KUKA KRL program: ps_p13060r5_msr_lta_c1.src, ps_p13060r5_msr_lta_c1.dat

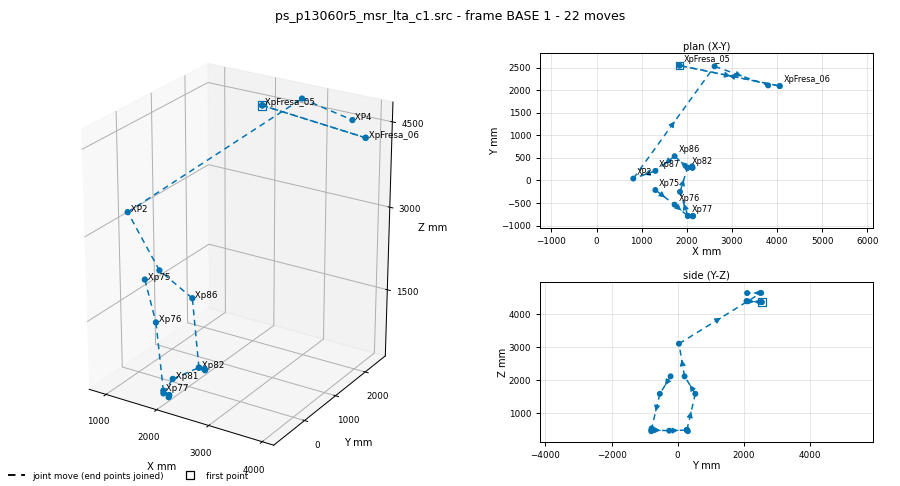
[picture p0: tool path of ps_p13060r5_msr_lta_c1.src in frame BASE 1, 22 of 24 moves have a stored position in this frame; points joined in program order, loops and branches not executed]
--- ps_p13060r5_msr_lta_c1.src ---
&ACCESS RVO
&REL 5
&COMMENT SOLDA MSR LTA GUN C1
&PARAM DISKPATH = KRC:\R1\Program
DEF ps_p13060r5_msr_lta_c1( )
;FOLD INI
  ;FOLD BASISTECH INI
    GLOBAL INTERRUPT DECL 3 WHEN $STOPMESS==TRUE DO IR_STOPM ( )
    INTERRUPT ON 3
    BAS (#INITMOV,0 )
  ;ENDFOLD (BASISTECH INI)
;FOLD SPOTTECH INI
USERSPOT(#INIT)
;ENDFOLD (SPOTTECH INI)
;FOLD GRIPPERTECH INI

;ENDFOLD (GRIPPERTECH INI)
  ;FOLD USER INI
    ;Make your modifications here

     ;FOLD COLLISION_V_3.01 INI ;%{E}
        IF (COLLISION_DATA[1].I_NR>0) THEN
          GLOBAL INTERRUPT DECL 21 WHEN $IN[COLLISION_DATA[1].I_NR]==FALSE DO COLLSTOP (1,0 )
        ENDIF
        IF (COLLISION_DATA[2].I_NR>0) THEN
          GLOBAL INTERRUPT DECL 22 WHEN $IN[COLLISION_DATA[2].I_NR]==FALSE DO COLLSTOP (2,0 )
        ENDIF
        IF (COLLISION_DATA[3].I_NR>0) THEN
          GLOBAL INTERRUPT DECL 23 WHEN $IN[COLLISION_DATA[3].I_NR]==FALSE DO COLLSTOP (3,0 )
        ENDIF
        IF (COLLISION_DATA[4].I_NR>0) THEN
          GLOBAL INTERRUPT DECL 24 WHEN $IN[COLLISION_DATA[4].I_NR]==FALSE DO COLLSTOP (4,0 )
        ENDIF
     ;ENDFOLD (Collision)

  ;ENDFOLD (USER INI)
;ENDFOLD (INI)

; Caracterização dos meios de produção: P13.060-R5
; Versão atual: 17/07/2013 Nome: Solda C1
; Change: MGS/LTA

chk_w2_wechs_ok ( )           ; VERIFICAÇÃO DE FERRAMENA: C1

;FOLD PTP HOME2 Vel=100 % DEFAULT;%{PE}%R 8.2.20,%MKUKATPBASIS,%CMOVE,%VPTP,%P 1:PTP, 2:HOME2, 3:, 5:100, 7:DEFAULT
$BWDSTART=FALSE
PDAT_ACT=PDEFAULT
FDAT_ACT=FHOME2
BAS(#PTP_PARAMS,100)
PTP XHOME2
;ENDFOLD

IF MaxStandMenge (1) THEN
 MaxStandmengeErreicht (1)
ENDIF

IF Elektrodenwechsel (1) THEN
;FOLD PTP pFresa_05 CONT Vel=100 % PDAT4 Tool[2]:Gun C1 Base[1]:Actros;%{PE}%R 8.2.20,%MKUKATPBASIS,%CMOVE,%VPTP,%P 1:PTP, 2:pFresa_05, 3:C_DIS, 5:100, 7:PDAT4
$BWDSTART=FALSE
PDAT_ACT=PPDAT4
FDAT_ACT=FpFresa_05
BAS(#PTP_PARAMS,100)
PTP XpFresa_05 C_DIS
;ENDFOLD
;FOLD PULSE 168 'DOCK 1 Fechar Proteção' State=TRUE Time=1 sec;%{PE}%R 8.2.20,%MKUKATPBASIS,%COUT,%VPULSE,%P 2:168, 3:DOCK 1 Fechar Proteção, 5:TRUE, 6:, 8:1
PULSE($OUT[168], TRUE,1)
;ENDFOLD
;FOLD WAIT FOR ( IN 166 'DOCK 1 Proteção Fechada' );%{PE}%R 8.2.20,%MKUKATPBASIS,%CEXT_WAIT_FOR,%VEXT_WAIT_FOR,%P 2:, 4:, 5:$IN, 6:166, 7:DOCK 1 Proteção Fechada, 9:
WAIT FOR  ( $IN[166] )
;ENDFOLD
;FOLD PTP pFresa_06 CONT Vel=100 % PDAT5 Tool[2]:Gun C1 Base[1]:Actros;%{PE}%R 8.2.20,%MKUKATPBASIS,%CMOVE,%VPTP,%P 1:PTP, 2:pFresa_06, 3:C_DIS, 5:100, 7:PDAT5
$BWDSTART=FALSE
PDAT_ACT=PPDAT5
FDAT_ACT=FpFresa_06
BAS(#PTP_PARAMS,100)
PTP XpFresa_06 C_DIS
;ENDFOLD
 e_Fraes_2 ()
;FOLD PTP pFresa_07 CONT Vel=100 % PDAT6 Tool[2]:Gun C1 Base[1]:Actros;%{PE}%R 8.2.20,%MKUKATPBASIS,%CMOVE,%VPTP,%P 1:PTP, 2:pFresa_07, 3:C_DIS, 5:100, 7:PDAT6
$BWDSTART=FALSE
PDAT_ACT=PPDAT6
FDAT_ACT=FpFresa_07
BAS(#PTP_PARAMS,100)
PTP XpFresa_07 C_DIS
;ENDFOLD
;FOLD PTP pFresa_08 CONT Vel=100 % PDAT7 Tool[2]:Gun C1 Base[1]:Actros;%{PE}%R 8.2.20,%MKUKATPBASIS,%CMOVE,%VPTP,%P 1:PTP, 2:pFresa_08, 3:C_DIS, 5:100, 7:PDAT7
$BWDSTART=FALSE
PDAT_ACT=PPDAT7
FDAT_ACT=FpFresa_08
BAS(#PTP_PARAMS,100)
PTP XpFresa_08 C_DIS
;ENDFOLD
ENDIF

;FOLD PTP HOME2 Vel=100 % DEFAULT;%{PE}%R 8.2.20,%MKUKATPBASIS,%CMOVE,%VPTP,%P 1:PTP, 2:HOME2, 3:, 5:100, 7:DEFAULT
$BWDSTART=FALSE
PDAT_ACT=PDEFAULT
FDAT_ACT=FHOME2
BAS(#PTP_PARAMS,100)
PTP XHOME2
;ENDFOLD

;FOLD OUT 3339 'R5 SOLDANDO' State=FALSE ;%{PE}%R 8.2.20,%MKUKATPBASIS,%COUT,%VOUTX,%P 2:3339, 3:R5 SOLDANDO, 5:FALSE, 6:
$OUT[3339]=FALSE
;ENDFOLD

;FOLD PTP p75 CONT Vel=100 % P_OLP2 Tool[2]:Gun C1 Base[1]:Actros;%{PE}%R 8.2.20,%MKUKATPBASIS,%CMOVE,%VPTP,%P 1:PTP, 2:p75, 3:C_DIS, 5:100, 7:P_OLP2
$BWDSTART=FALSE
PDAT_ACT=PP_OLP2
FDAT_ACT=Fp75
BAS(#PTP_PARAMS,100)
PTP Xp75 C_DIS
;ENDFOLD
;FOLD PTP p76 CONT Vel=100 % P_OLP3 Tool[2]:Gun C1 Base[1]:Actros;%{PE}%R8.2,%MKUKATPBASIS,%CMOVE,%VPTP,%P 1:PTP, 2:p76, 3:C_DIS, 5:100, 7:P_OLP3
$BWDSTART = FALSE
PDAT_ACT= PP_OLP3
FDAT_ACT= Fp76
BAS(#PTP_PARAMS,100)
PTP Xp76 C_DIS
;ENDFOLD
;FOLD PTP p77 CONT Vel=100 % P_OLP4 Tool[2]:Gun C1 Base[1]:Actros;%{PE}%R8.2,%MKUKATPBASIS,%CMOVE,%VPTP,%P 1:PTP, 2:p77, 3:C_DIS, 5:100, 7:P_OLP4
$BWDSTART = FALSE
PDAT_ACT= PP_OLP4
FDAT_ACT= Fp77
BAS(#PTP_PARAMS,100)
PTP Xp77 C_DIS
;ENDFOLD
;FOLD PTP p78 CONT Vel=100 % P_OLP5 Tool[2]:Gun C1 Base[1]:Actros;%{PE}%R8.2,%MKUKATPBASIS,%CMOVE,%VPTP,%P 1:PTP, 2:p78, 3:C_DIS, 5:100, 7:P_OLP5
$BWDSTART = FALSE
PDAT_ACT= PP_OLP5
FDAT_ACT= Fp78
BAS(#PTP_PARAMS,100)
PTP Xp78 C_DIS
;ENDFOLD

;FOLD ; SWP_60_5471;%{PE}%R8.2,%MKUKATPBASIS,%CCOMMENT,%VNORMAL,%P 2: SWP_60_5471
;ENDFOLD
;FOLD PTP swp_60_5471 P_OLP6 SPOT Gun=1 RETR OPN PgNo1=55 ACTIVE=1 Tool[2]:Gun C1 Base[1]:Actros;%{PE}%R 8.2.2,%MKUKATPSPOT,%CSPOT,%VPTP,%P 1:PTP, 2:swp_60_5471, 3:, 5:100, 7:P_OLP6, 10:1, 12:#FIRST, 14:#OPN, 16:55, 18:1, 20:1, 22:0, 24:1, 25:S_OLP1
$BWDSTART=FALSE
PDAT_ACT=PP_OLP6
FDAT_ACT=Fswp_60_5471
BAS(#PTP_PARAMS,PP_OLP6.VEL)
S_ACT.GUN=1
S_ACT.PAIR=SDEFAULT.PAIR
S_ACT.RETR=#OPN
S_ACT.CLO_TM=1
S_ACT.PGNO1=55
S_ACT.PGNO2=SDEFAULT.PGNO2
S_ACT.PRESS1=SDEFAULT.PRESS1
S_ACT.PRESS2=SDEFAULT.PRESS2
S_READY=FALSE
PTP Xswp_60_5471
USERSPOT(#SPOT, S_ACT)
WAIT FOR S_READY
;ENDFOLD

;FOLD PTP p79 CONT Vel=100 % P_OLP7 Tool[2]:Gun C1 Base[1]:Actros;%{PE}%R8.2,%MKUKATPBASIS,%CMOVE,%VPTP,%P 1:PTP, 2:p79, 3:C_DIS, 5:100, 7:P_OLP7
$BWDSTART = FALSE
PDAT_ACT= PP_OLP7
FDAT_ACT= Fp79
BAS(#PTP_PARAMS,100)
PTP Xp79 C_DIS
;ENDFOLD
;FOLD PTP p80 CONT Vel=100 % P_OLP8 Tool[2]:Gun C1 Base[1]:Actros;%{PE}%R8.2,%MKUKATPBASIS,%CMOVE,%VPTP,%P 1:PTP, 2:p80, 3:C_DIS, 5:100, 7:P_OLP8
$BWDSTART = FALSE
PDAT_ACT= PP_OLP8
FDAT_ACT= Fp80
BAS(#PTP_PARAMS,100)
PTP Xp80 C_DIS
;ENDFOLD
;FOLD PTP p81 CONT Vel=100 % P_OLP9 Tool[2]:Gun C1 Base[1]:Actros;%{PE}%R8.2,%MKUKATPBASIS,%CMOVE,%VPTP,%P 1:PTP, 2:p81, 3:C_DIS, 5:100, 7:P_OLP9
$BWDSTART = FALSE
PDAT_ACT= PP_OLP9
FDAT_ACT= Fp81
BAS(#PTP_PARAMS,100)
PTP Xp81 C_DIS
;ENDFOLD
;FOLD PTP p82 CONT Vel=100 % P_OLP10 Tool[2]:Gun C1 Base[1]:Actros;%{PE}%R8.2,%MKUKATPBASIS,%CMOVE,%VPTP,%P 1:PTP, 2:p82, 3:C_DIS, 5:100, 7:P_OLP10
$BWDSTART = FALSE
PDAT_ACT= PP_OLP10
FDAT_ACT= Fp82
BAS(#PTP_PARAMS,100)
PTP Xp82 C_DIS
;ENDFOLD
;FOLD PTP p83 CONT Vel=100 % P_OLP11 Tool[2]:Gun C1 Base[1]:Actros;%{PE}%R8.2,%MKUKATPBASIS,%CMOVE,%VPTP,%P 1:PTP, 2:p83, 3:C_DIS, 5:100, 7:P_OLP11
$BWDSTART = FALSE
PDAT_ACT= PP_OLP11
FDAT_ACT= Fp83
BAS(#PTP_PARAMS,100)
PTP Xp83 C_DIS
;ENDFOLD

;FOLD ; SWP_60_5452;%{PE}%R8.2,%MKUKATPBASIS,%CCOMMENT,%VNORMAL,%P 2: SWP_60_5452
;ENDFOLD
;FOLD PTP swp_60_5452 P_OLP12 SPOT Gun=1 RETR OPN PgNo1=56 ACTIVE=1 Tool[2]:Gun C1 Base[1]:Actros;%{PE}%R 8.2.2,%MKUKATPSPOT,%CSPOT,%VPTP,%P 1:PTP, 2:swp_60_5452, 3:, 5:100, 7:P_OLP12, 10:1, 12:#FIRST, 14:#OPN, 16:56, 18:1, 20:1, 22:0, 24:1, 25:S_OLP2
$BWDSTART=FALSE
PDAT_ACT=PP_OLP12
FDAT_ACT=Fswp_60_5452
BAS(#PTP_PARAMS,PP_OLP12.VEL)
S_ACT.GUN=1
S_ACT.PAIR=SDEFAULT.PAIR
S_ACT.RETR=#OPN
S_ACT.CLO_TM=1
S_ACT.PGNO1=56
S_ACT.PGNO2=SDEFAULT.PGNO2
S_ACT.PRESS1=SDEFAULT.PRESS1
S_ACT.PRESS2=SDEFAULT.PRESS2
S_READY=FALSE
PTP Xswp_60_5452
USERSPOT(#SPOT, S_ACT)
WAIT FOR S_READY
;ENDFOLD

;FOLD PTP p84 CONT Vel=100 % P_OLP13 Tool[2]:Gun C1 Base[1]:Actros;%{PE}%R8.2,%MKUKATPBASIS,%CMOVE,%VPTP,%P 1:PTP, 2:p84, 3:C_DIS, 5:100, 7:P_OLP13
$BWDSTART = FALSE
PDAT_ACT= PP_OLP13
FDAT_ACT= Fp84
BAS(#PTP_PARAMS,100)
PTP Xp84 C_DIS
;ENDFOLD
;FOLD PTP p85 CONT Vel=100 % P_OLP14 Tool[2]:Gun C1 Base[1]:Actros;%{PE}%R8.2,%MKUKATPBASIS,%CMOVE,%VPTP,%P 1:PTP, 2:p85, 3:C_DIS, 5:100, 7:P_OLP14
$BWDSTART = FALSE
PDAT_ACT= PP_OLP14
FDAT_ACT= Fp85
BAS(#PTP_PARAMS,100)
PTP Xp85 C_DIS
;ENDFOLD
;FOLD PTP p86 CONT Vel=100 % P_OLP15 Tool[2]:Gun C1 Base[1]:Actros;%{PE}%R8.2,%MKUKATPBASIS,%CMOVE,%VPTP,%P 1:PTP, 2:p86, 3:C_DIS, 5:100, 7:P_OLP15
$BWDSTART = FALSE
PDAT_ACT= PP_OLP15
FDAT_ACT= Fp86
BAS(#PTP_PARAMS,100)
PTP Xp86 C_DIS
;ENDFOLD
;FOLD PTP p87 CONT Vel=100 % P_OLP16 Tool[2]:Gun C1 Base[1]:Actros;%{PE}%R8.2,%MKUKATPBASIS,%CMOVE,%VPTP,%P 1:PTP, 2:p87, 3:C_DIS, 5:100, 7:P_OLP16
$BWDSTART = FALSE
PDAT_ACT= PP_OLP16
FDAT_ACT= Fp87
BAS(#PTP_PARAMS,100)
PTP Xp87 C_DIS
;ENDFOLD

;FOLD OUT 3339 'R5 SOLDANDO' State=TRUE CONT;%{PE}%R 8.2.20,%MKUKATPBASIS,%COUT,%VOUTX,%P 2:3339, 3:R5 SOLDANDO, 5:TRUE, 6:CONTINUE
CONTINUE
$OUT[3339]=TRUE
;ENDFOLD

;FOLD PTP P2 CONT Vel=100 % PDAT2 Tool[2]:Gun C1 Base[1]:Actros;%{PE}%R 8.2.20,%MKUKATPBASIS,%CMOVE,%VPTP,%P 1:PTP, 2:P2, 3:C_DIS, 5:100, 7:PDAT2
$BWDSTART=FALSE
PDAT_ACT=PPDAT2
FDAT_ACT=FP2
BAS(#PTP_PARAMS,100)
PTP XP2 C_DIS
;ENDFOLD
;FOLD PTP P3 CONT Vel=100 % PDAT3 Tool[2]:Gun C1 Base[1]:Actros;%{PE}%R 8.2.20,%MKUKATPBASIS,%CMOVE,%VPTP,%P 1:PTP, 2:P3, 3:C_DIS, 5:100, 7:PDAT3
$BWDSTART=FALSE
PDAT_ACT=PPDAT3
FDAT_ACT=FP3
BAS(#PTP_PARAMS,100)
PTP XP3 C_DIS
;ENDFOLD
;FOLD PTP P4 Vel=100 % PDAT8 Tool[2]:Gun C1 Base[1]:Actros;%{PE}%R 8.2.20,%MKUKATPBASIS,%CMOVE,%VPTP,%P 1:PTP, 2:P4, 3:, 5:100, 7:PDAT8
$BWDSTART=FALSE
PDAT_ACT=PPDAT8
FDAT_ACT=FP4
BAS(#PTP_PARAMS,100)
PTP XP4
;ENDFOLD

IF FraesAnf (1) THEN

 f_Fraes_2()

ENDIF

END

--- ps_p13060r5_msr_lta_c1.dat ---
&ACCESS RVO
&REL 5
&COMMENT SOLDA MSR LTA GUN C1
&PARAM DISKPATH = KRC:\R1\Program
DEFDAT  ps_p13060r5_msr_lta_c1
;FOLD EXTERNAL DECLARATIONS;%{PE}%MKUKATPBASIS,%CEXT,%VCOMMON,%P
;FOLD GRIPPERTECH EXT
EXT  H50 (INT  :IN,INT  :IN,INT  :IN,GRP_TYP  :IN )
;ENDFOLD (GRIPPERTECH EXT)
;FOLD SPOTTECH EXT
EXT  USERSPOT (S_COMMAND  :IN,SPOT_TYPE  :IN )
;ENDFOLD (SPOTTECH EXT)
;FOLD BASISTECH EXT;%{PE}%MKUKATPBASIS,%CEXT,%VEXT,%P
EXT  BAS (BAS_COMMAND  :IN,REAL  :IN )
DECL INT SUCCESS
;ENDFOLD (BASISTECH EXT)
;FOLD USER EXT;%{E}%MKUKATPUSER,%CEXT,%VEXT,%P
;Make your modifications here

;ENDFOLD (USER EXT)
;ENDFOLD (EXTERNAL DECLARATIONS)

;# ============ START PATH : swp_p13060r5_msr_lta_c1 =============
DECL FDAT Fp75={TOOL_NO 2,BASE_NO 1,IPO_FRAME #BASE,POINT2[] " "}
DECL PDAT PP_OLP2={VEL 100.0,ACC 100.0,APO_DIST 100.0,APO_MODE #CDIS}
DECL E6POS Xp75={X 1303.604,Y -211.761002,Z 2118.72705,A -126.906303,B 65.6848984,C 49.8302002,S 2,T 10}
DECL FDAT Fp76={TOOL_NO 2,BASE_NO 1,IPO_FRAME #BASE,POINT2[] " "}
DECL PDAT PP_OLP3={VEL 100.0,ACC 100.0,APO_DIST 100.0,APO_MODE #CDIS}
DECL E6POS Xp76={X 1729.96497,Y -537.172974,Z 1590.30103,A -75.8211975,B 62.4005013,C 105.7089,S 2,T 11}
DECL FDAT Fp77={TOOL_NO 2,BASE_NO 1,IPO_FRAME #BASE,POINT2[] " "}
DECL PDAT PP_OLP4={VEL 100.0,ACC 100.0,APO_DIST 100.0,APO_MODE #CDIS}
DECL E6POS Xp77={X 2022.47803,Y -785.769104,Z 542.154907,A -89.9998932,B 70.0002136,C 89.9999771,S 2,T 9,E1 0.0,E2 0.0,E3 0.0,E4 0.0,E5 0.0,E6 0.0}
DECL FDAT Fp78={TOOL_NO 2,BASE_NO 1,IPO_FRAME #BASE,POINT2[] " "}
DECL PDAT PP_OLP5={VEL 100.0,ACC 100.0,APO_DIST 100.0,APO_MODE #CDIS}
DECL E6POS Xp78={X 2134.76611,Y -787.281006,Z 490.900208,A -89.9603119,B 69.9023438,C 90.0867233,S 2,T 9,E1 0.0,E2 0.0,E3 0.0,E4 0.0,E5 0.0,E6 0.0}
DECL FDAT Fswp_60_5471={TOOL_NO 2,BASE_NO 1,IPO_FRAME #BASE,POINT2[] " "}
DECL PDAT PP_OLP6={VEL 100.0,ACC 100.0,APO_DIST 0.0}
DECL SPOT_TYPE SS_OLP1={GUN 2,PAIR #FIRST,RETR #CLO,CLO_TM 0,PGNO1 1,PRESS1 1.0,PGNO2 0,PRESS2 0.0}
DECL E6POS Xswp_60_5471={X 2130.88208,Y -795.672913,Z 457.943512,A -90.164978,B 69.9813766,C 89.8283234,S 2,T 9,E1 0.0,E2 0.0,E3 0.0,E4 0.0,E5 0.0,E6 0.0}
DECL FDAT Fp79={TOOL_NO 2,BASE_NO 1,IPO_FRAME #BASE,POINT2[] " "}
DECL PDAT PP_OLP7={VEL 100.0,ACC 100.0,APO_DIST 100.0,APO_MODE #CDIS}
DECL E6POS Xp79={X 2134.00098,Y -785.97699,Z 492.528015,A -90.0,B 70.0,C 90.0,S 2,T 9,E1 0.0,E2 0.0,E3 0.0,E4 0.0,E5 0.0,E6 0.0}
DECL FDAT Fp80={TOOL_NO 2,BASE_NO 1,IPO_FRAME #BASE,POINT2[] " "}
DECL PDAT PP_OLP8={VEL 100.0,ACC 100.0,APO_DIST 100.0,APO_MODE #CDIS}
DECL E6POS Xp80={X 2023.00098,Y -785.97699,Z 492.527008,A -90.0,B 70.0,C 90.0,S 2,T 9}
DECL FDAT Fp81={TOOL_NO 2,BASE_NO 1,IPO_FRAME #BASE,POINT2[] " "}
DECL PDAT PP_OLP9={VEL 100.0,ACC 100.0,APO_DIST 100.0,APO_MODE #CDIS}
DECL E6POS Xp81={X 1849.08496,Y -251.766006,Z 473.174011,A -153.737396,B 79.8789978,C 25.6958008,S 2,T 9}
DECL FDAT Fp82={TOOL_NO 2,BASE_NO 1,IPO_FRAME #BASE,POINT2[] " "}
DECL PDAT PP_OLP10={VEL 100.0,ACC 100.0,APO_DIST 100.0,APO_MODE #CDIS}
DECL E6POS Xp82={X 2015.50195,Y 281.194,Z 494.32901,A 90.0,B 65.0,C -90.0,S 2,T 33}
DECL FDAT Fp83={TOOL_NO 2,BASE_NO 1,IPO_FRAME #BASE,POINT2[] " "}
DECL PDAT PP_OLP11={VEL 100.0,ACC 100.0,APO_DIST 100.0,APO_MODE #CDIS}
DECL E6POS Xp83={X 2125.00098,Y 281.194,Z 494.32901,A 90.0,B 65.0,C -90.0,S 2,T 33}
DECL FDAT Fswp_60_5452={TOOL_NO 2,BASE_NO 1,IPO_FRAME #BASE,POINT2[] " "}
DECL PDAT PP_OLP12={VEL 100.0,ACC 100.0,APO_DIST 0.0}
DECL SPOT_TYPE SS_OLP2={GUN 1,PAIR #FIRST,RETR #CLO,CLO_TM 0,PGNO1 1,PRESS1 1.0,PGNO2 0,PRESS2 0.0}
DECL E6POS Xswp_60_5452={X 2116.53296,Y 312.069702,Z 459.115387,A 89.9984131,B 64.9997482,C -90.001503,S 2,T 33,E1 0.0,E2 0.0,E3 0.0,E4 0.0,E5 0.0,E6 0.0}
DECL FDAT Fp84={TOOL_NO 2,BASE_NO 1,IPO_FRAME #BASE,POINT2[] " "}
DECL PDAT PP_OLP13={VEL 100.0,ACC 100.0,APO_DIST 100.0,APO_MODE #CDIS}
DECL E6POS Xp84={X 2125.00098,Y 281.194,Z 494.32901,A 90.0,B 65.0,C -90.0,S 2,T 33}
DECL FDAT Fp85={TOOL_NO 2,BASE_NO 1,IPO_FRAME #BASE,POINT2[] " "}
DECL PDAT PP_OLP14={VEL 100.0,ACC 100.0,APO_DIST 100.0,APO_MODE #CDIS}
DECL E6POS Xp85={X 2015.50195,Y 281.194,Z 494.32901,A 90.0,B 65.0,C -90.0,S 2,T 33}
DECL FDAT Fp86={TOOL_NO 2,BASE_NO 1,IPO_FRAME #BASE,POINT2[] " "}
DECL PDAT PP_OLP15={VEL 100.0,ACC 100.0,APO_DIST 100.0,APO_MODE #CDIS}
DECL E6POS Xp86={X 1729.96497,Y 537.172974,Z 1590.30103,A 75.8211975,B 62.4005013,C -105.7089,S 2,T 34}
DECL FDAT Fp87={TOOL_NO 2,BASE_NO 1,IPO_FRAME #BASE,POINT2[] " "}
DECL PDAT PP_OLP16={VEL 100.0,ACC 100.0,APO_DIST 100.0,APO_MODE #CDIS}
DECL E6POS Xp87={X 1303.604,Y 211.761002,Z 2118.72705,A 126.906303,B 65.6848984,C -49.8302002,S 2,T 35}
DECL PDAT PPDAT2={VEL 100.0,ACC 100.0,APO_DIST 100.0,APO_MODE #CDIS}
DECL E6POS XP2={X 814.124023,Y 41.7988205,Z 3106.80688,A -178.988297,B 40.6093292,C 0.315527499,S 2,T 2,E1 0.0,E2 0.0,E3 0.0,E4 0.0,E5 0.0,E6 0.0}
DECL FDAT FP2={TOOL_NO 2,BASE_NO 1,IPO_FRAME #BASE,POINT2[] " "}
DECL PDAT PPDAT3={VEL 100.0,ACC 100.0,APO_DIST 100.0,APO_MODE #CDIS}
DECL E6POS XP3={X 2614.91089,Y 2529.12793,Z 4644.24902,A 61.9992714,B -36.66222,C 37.742569,S 2,T 42,E1 0.0,E2 0.0,E3 0.0,E4 0.0,E5 0.0,E6 0.0}
DECL FDAT FP3={TOOL_NO 2,BASE_NO 1,IPO_FRAME #BASE,POINT2[] " ",TQ_STATE FALSE}
DECL SPOT_SUGG_T LAST_SPOT={GUN[] "1                       ",RETR_CMD[] "#OPN                    ",CHOISE[] "#FIRST                  ",CLO_TM[] "0                       ",PGNO1[] "1                       ",PRESS1[] "0                       ",PGNO2[] "1                       ",PRESS2[] "0                       ",SPOT_PARAMS[] "NORMAL                  "}
DECL FDAT FHOME2={TOOL_NO 0,BASE_NO 0,IPO_FRAME #BASE,POINT2[] " ",TQ_STATE FALSE}
DECL PDAT PPDAT4={VEL 100.0,ACC 100.0,APO_DIST 100.0,APO_MODE #CDIS}
DECL E6POS XpFresa_05={X 1838.66003,Y 2546.56006,Z 4367.69092,A 105.045502,B -33.6448593,C -0.634051323,S 2,T 2,E1 0.0,E2 0.0,E3 0.0,E4 0.0,E5 0.0,E6 0.0}
DECL FDAT FpFresa_05={TOOL_NO 2,BASE_NO 1,IPO_FRAME #BASE,POINT2[] " ",TQ_STATE FALSE}
DECL PDAT PPDAT5={VEL 100.0,ACC 100.0,APO_DIST 100.0,APO_MODE #CDIS}
DECL E6POS XpFresa_06={X 4058.65503,Y 2091.6001,Z 4393.26904,A 52.5592613,B -34.2167282,C -0.74924773,S 2,T 2,E1 0.0,E2 0.0,E3 0.0,E4 0.0,E5 0.0,E6 0.0}
DECL FDAT FpFresa_06={TOOL_NO 2,BASE_NO 1,IPO_FRAME #BASE,POINT2[] " ",TQ_STATE FALSE}
DECL PDAT PPDAT6={VEL 100.0,ACC 100.0,APO_DIST 100.0,APO_MODE #CDIS}
DECL E6POS XpFresa_07={X 4058.65503,Y 2091.6001,Z 4393.26904,A 52.5592613,B -34.2167282,C -0.74924773,S 2,T 2,E1 0.0,E2 0.0,E3 0.0,E4 0.0,E5 0.0,E6 0.0}
DECL FDAT FpFresa_07={TOOL_NO 2,BASE_NO 1,IPO_FRAME #BASE,POINT2[] " ",TQ_STATE FALSE}
DECL PDAT PPDAT7={VEL 100.0,ACC 100.0,APO_DIST 100.0,APO_MODE #CDIS}
DECL E6POS XpFresa_08={X 1838.66003,Y 2546.56006,Z 4367.69092,A 105.045502,B -33.6448593,C -0.634051323,S 2,T 2,E1 0.0,E2 0.0,E3 0.0,E4 0.0,E5 0.0,E6 0.0}
DECL FDAT FpFresa_08={TOOL_NO 2,BASE_NO 1,IPO_FRAME #BASE,POINT2[] " ",TQ_STATE FALSE}
DECL E6POS XP4={X 3802.31104,Y 2105.88989,Z 4640.2832,A 19.5630798,B -23.7333107,C 61.6030312,S 2,T 42,E1 0.0,E2 0.0,E3 0.0,E4 0.0,E5 0.0,E6 0.0}
DECL FDAT FP4={TOOL_NO 2,BASE_NO 1,IPO_FRAME #BASE,POINT2[] " ",TQ_STATE FALSE}
DECL PDAT PPDAT8={VEL 100.0,ACC 100.0,APO_DIST 5.0,APO_MODE #CDIS}
ENDDAT
